FUNCTION UpdateEventTimeStampWithSystemTime
VAR_INPUT
	stEvent : REFERENCE TO ST_Event;
END_VAR
VAR
fbGETSYSTEMTIME : GETSYSTEMTIME;


stFileTime : T_FILETIME;

END_VAR

fbGETSYSTEMTIME(timeLoDW => stFileTime.dwLowDateTime , 
				timeHiDW => stFileTime.dwHighDateTime);
				
stEvent.dtTimestamp := FILETIME_TO_DT(fileTime := stFileTime);

END_FUNCTION

(* stored: Version 1.1.0.1, ProductVersion 3.1.4024.12
   POU UpdateEventTimeStampWithSystemTime: Id {3d5b7336-b492-45ee-9bc3-4633563c28e5}, SpecialFunc None *)
